PROGRAM PropValve
VAR
	mcPower	:	MC_Power;
	stPropValve	:	ST_PropValveMKS253;
	tofLLSFilter	:	TOF := (PT:=T#100MS);
	tofHLSFilter	:	TOF := (PT:=T#100MS);
END_VAR

(* The low limit switch was flakey, I added the filters*)
tofLLSFilter(IN:=stPropValve.i_LLS);
tofHLSFilter(IN:=stPropValve.i_HLS);
mcPower.Enable_Positive := tofHLSFilter.Q;
mcPower.Enable_Negative := tofLLSFilter.Q;
mcPower(Axis:=stPropValve.stAxis);

END_PROGRAM

(* stored: Version 1.1.0.1, ProductVersion 3.1.4020.12
   POU PropValve: Id {5d37ea8b-affd-40c7-9959-7bc359f6de15}, SpecialFunc None *)
